FUNCTION_BLOCK FB_RecipeBuilderRectangle EXTENDS FB_RecipeBase

METHOD Build : BOOL
VAR_INST
    TotalY          : REAL;
    TotalX          : REAL;
    ShorterY        : REAL;
    ShorterX        : REAL;
END_VAR
_Busy := TRUE;
_Done := FALSE;
_Error := FALSE;
Build := FALSE;
THIS^.UpdateNestingLimits();

// 2. Jeśli detal wystaje poza maszynę - przerywamy od razu!
IF NOT _Config.IsValid THEN
    _Busy := FALSE;
    _Error := TRUE; 
    Build := FALSE;
    RETURN;
END_IF
// 3. Pobieramy wyliczone gabaryty nominalne do lokalnych zmiennych roboczych
TotalX   := _NominalX;
TotalY   := _NominalY; 

// ------------------------------------
// 1. Segregracja frezowania (Grooving)
// ------------------------------------
_SegmentsToGroove := 0;
     
// ------------------------------------
// 2. Cięcie w osi X (Cut X)
// ------------------------------------+ 
_SegmentsToCutX := 2;

// Short Box Segments
_SegmentsCutX[1].Start.X := TotalX + _Config.CuttingOverpass;
_SegmentsCutX[1].Stop.X  := -_Config.CuttingOverpass;
_SegmentsCutX[1].Start.Y := 0;
_SegmentsCutX[1].Stop.Y  := 0;        

_SegmentsCutX[2].Start.X := TotalX + _Config.CuttingOverpass;                         
_SegmentsCutX[2].Stop.X  := - _Config.CuttingOverpass;                          
_SegmentsCutX[2].Start.Y := TotalY;
_SegmentsCutX[2].Stop.Y  := TotalY;        

// ------------------------------------
// 3. Cięcie w osi Y (Cut Y)
// ------------------------------------
_SegmentsToCutY := 2;

// Short Box Segments
_SegmentsCutY[1].Start.X := 0;                               
_SegmentsCutY[1].Stop.X  := 0;                               
_SegmentsCutY[1].Start.Y := TotalY +_Config.CuttingOverpass; 
_SegmentsCutY[1].Stop.Y  := -_Config.CuttingOverpass;        

_SegmentsCutY[2].Start.X := TotalX;                          
_SegmentsCutY[2].Stop.X  := TotalX;                          
_SegmentsCutY[2].Start.Y := TotalY +_Config.CuttingOverpass; 
_SegmentsCutY[2].Stop.Y  := -_Config.CuttingOverpass;        

_Busy := FALSE;
_Done := TRUE;
Build := TRUE;
END_METHOD

METHOD PROTECTED CalculateFootprint
VAR_INPUT
END_VAR
_NominalX := _Config.PanelFrontWidth;
_NominalY := _Config.PanelFrontLength;
END_METHOD

PROPERTY ExecutionRoute : E_ExecutionRoute
GET
ExecutionRoute := E_ExecutionRoute.ePTP;
END_GET
END_PROPERTY

METHOD FB_init : BOOL
VAR_INPUT
	bInitRetains : BOOL; // if TRUE, the retain variables are initialized (warm start / cold start)
	bInCopyCode : BOOL;  // if TRUE, the instance afterwards gets moved into the copy code (online change)
END_VAR
_Limits.PanelFrontLength.MinVal := 12.0;
_Limits.PanelFrontLength.MaxVal := 2400.0;

_Limits.PanelFrontWidth.MinVal  := 12.0;
_Limits.PanelFrontWidth.MaxVal  := 1200.0;

_Limits.PanelHeight.MinVal      := 12.0;
_Limits.PanelHeight.MaxVal      := 1234.0;

_Limits.RailHeightCorrection.MinVal := 12.0;
_Limits.RailHeightCorrection.MaxVal := 13.0;

_Limits.CuttingOverpass.MinVal := 0.0;
_Limits.CuttingOverpass.MaxVal := 50.0;

_Limits.GroovingOverpass.MinVal := 0.0;
_Limits.GroovingOverpass.MaxVal := 50.0;

_Limits.GrooveDepthZ.MinVal := 0.0;
_Limits.GrooveDepthZ.MaxVal := 9.0; //
END_METHOD

END_FUNCTION_BLOCK

(* stored: Version 1.1.0.1, ProductVersion 3.1.4024.15
   POU FB_RecipeBuilderRectangle: Id {6c4812e0-2124-4ebf-9425-648a799633b0}, SpecialFunc None
   Method Build: Id {383e92b6-e22e-4900-a8ba-78049e770f6e}
   Method CalculateFootprint: Id {b115e399-8fb8-44ec-a54a-a3f7957f2856}
   Property ExecutionRoute: Id {5de48596-9966-4044-9349-927935ea8a70}
   Get Get: Id {70e41018-2eab-4116-a6c6-e2cc04c50b69}
   Method FB_init: Id {ee63f777-622f-4528-bf37-252b5ad994fe} *)
